Staubli VAL3: VelocityAddon.dtx

mdesc mNomSpeed
bool bSync
mdesc mNominal = {tmax=100, rmax=100, leave=1, reach=1, blend=cartesian}
tool tTool = {fatherId=flange[0], ioLink=valve1}
num nVelCmd[6]
num nMoveType
